PROGRAM POU
VAR
	fb : FB_ModbusMaster_PcCOM;
	fbb : FB_ModbusRtuMaster_KL6x22B;
	fbc : FB_ModbusRtuMaster_KL6x5B;
	tcpSlave : FB_ModbusSlaveTcp;
	tcpMaster : FB_ModbusMasterTcpIp;
END_VAR

END_PROGRAM

(* stored: Version 1.1.0.1, ProductVersion 3.1.4024.12
   POU POU: Id {e2653010-59d5-49c6-bdd0-b9433cd60d45}, SpecialFunc None *)
